FUNCTION_BLOCK sequence_T_08_loop (* Sequence with 8 Outputs looped, Transition by TIME *)
  (* Standard: 61499-2; Description: Copyright (c) 2024 HR Agrartechnik GmbH This program and the accompanying materials are made available under the terms of the Eclipse Public License 2.0 which is available at https://www.eclipse.org/legal/epl-2.0/ SPDX-License-Identifier: EPL-2.0 *)
  (* Version 1.0, 2024-03-02, Franz Höpfinger, HR Agrartechnik GmbH *)
  PACKAGE logiBUS::utils::sequence::timed;
  IMPORT logiBUS::utils::sequence::const::sequence;
  IMPORT logiBUS::utils::sequence::const::sequence::NO_TIME;
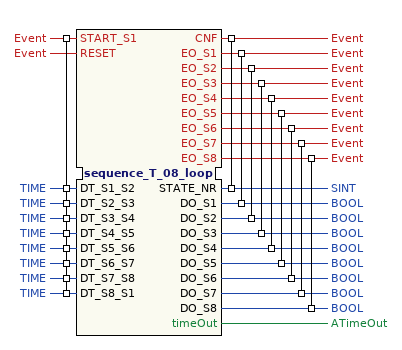
  EVENT_INPUT
    START_S1 WITH DT_S1_S2, DT_S2_S3, DT_S3_S4, DT_S4_S5, DT_S5_S6, DT_S6_S7, DT_S7_S8, DT_S8_S1; (* jump from START to State_01 *)
    RESET; (* Reset from any State to START *)
  END_EVENT
  EVENT_OUTPUT
    CNF WITH STATE_NR; (* Execution Confirmation *)
    EO_S1 WITH DO_S1;
    EO_S2 WITH DO_S2;
    EO_S3 WITH DO_S3;
    EO_S4 WITH DO_S4;
    EO_S5 WITH DO_S5;
    EO_S6 WITH DO_S6;
    EO_S7 WITH DO_S7;
    EO_S8 WITH DO_S8;
  END_EVENT
  VAR_INPUT
    DT_S1_S2 : TIME := NO_TIME; (* State_01 to State_02 timed *)
    DT_S2_S3 : TIME := NO_TIME; (* State_02 to State_03 timed *)
    DT_S3_S4 : TIME := NO_TIME; (* State_03 to State_04 timed *)
    DT_S4_S5 : TIME := NO_TIME; (* State_04 to State_05 timed *)
    DT_S5_S6 : TIME := NO_TIME; (* State_05 to State_06 timed *)
    DT_S6_S7 : TIME := NO_TIME; (* State_06 to State_07 timed *)
    DT_S7_S8 : TIME := NO_TIME; (* State_07 to State_08 timed *)
    DT_S8_S1 : TIME := NO_TIME; (* State_08 to State_01 timed *)
  END_VAR
  VAR_OUTPUT
    STATE_NR : SINT; (* State Number, START = 0, State_01 = 1 and so on. *)
    DO_S1 : BOOL; (* Output if State_01 is active *)
    DO_S2 : BOOL; (* Output if State_02 is active *)
    DO_S3 : BOOL; (* Output if State_03 is active *)
    DO_S4 : BOOL; (* Output if State_04 is active *)
    DO_S5 : BOOL; (* Output if State_05 is active *)
    DO_S6 : BOOL; (* Output if State_05 is active *)
    DO_S7 : BOOL; (* Output if State_05 is active *)
    DO_S8 : BOOL; (* Output if State_05 is active *)
  END_VAR
  PLUGS
    timeOut : iec61499::events::ATimeOut; (* timeOut Adapter *)
  END_PLUGS
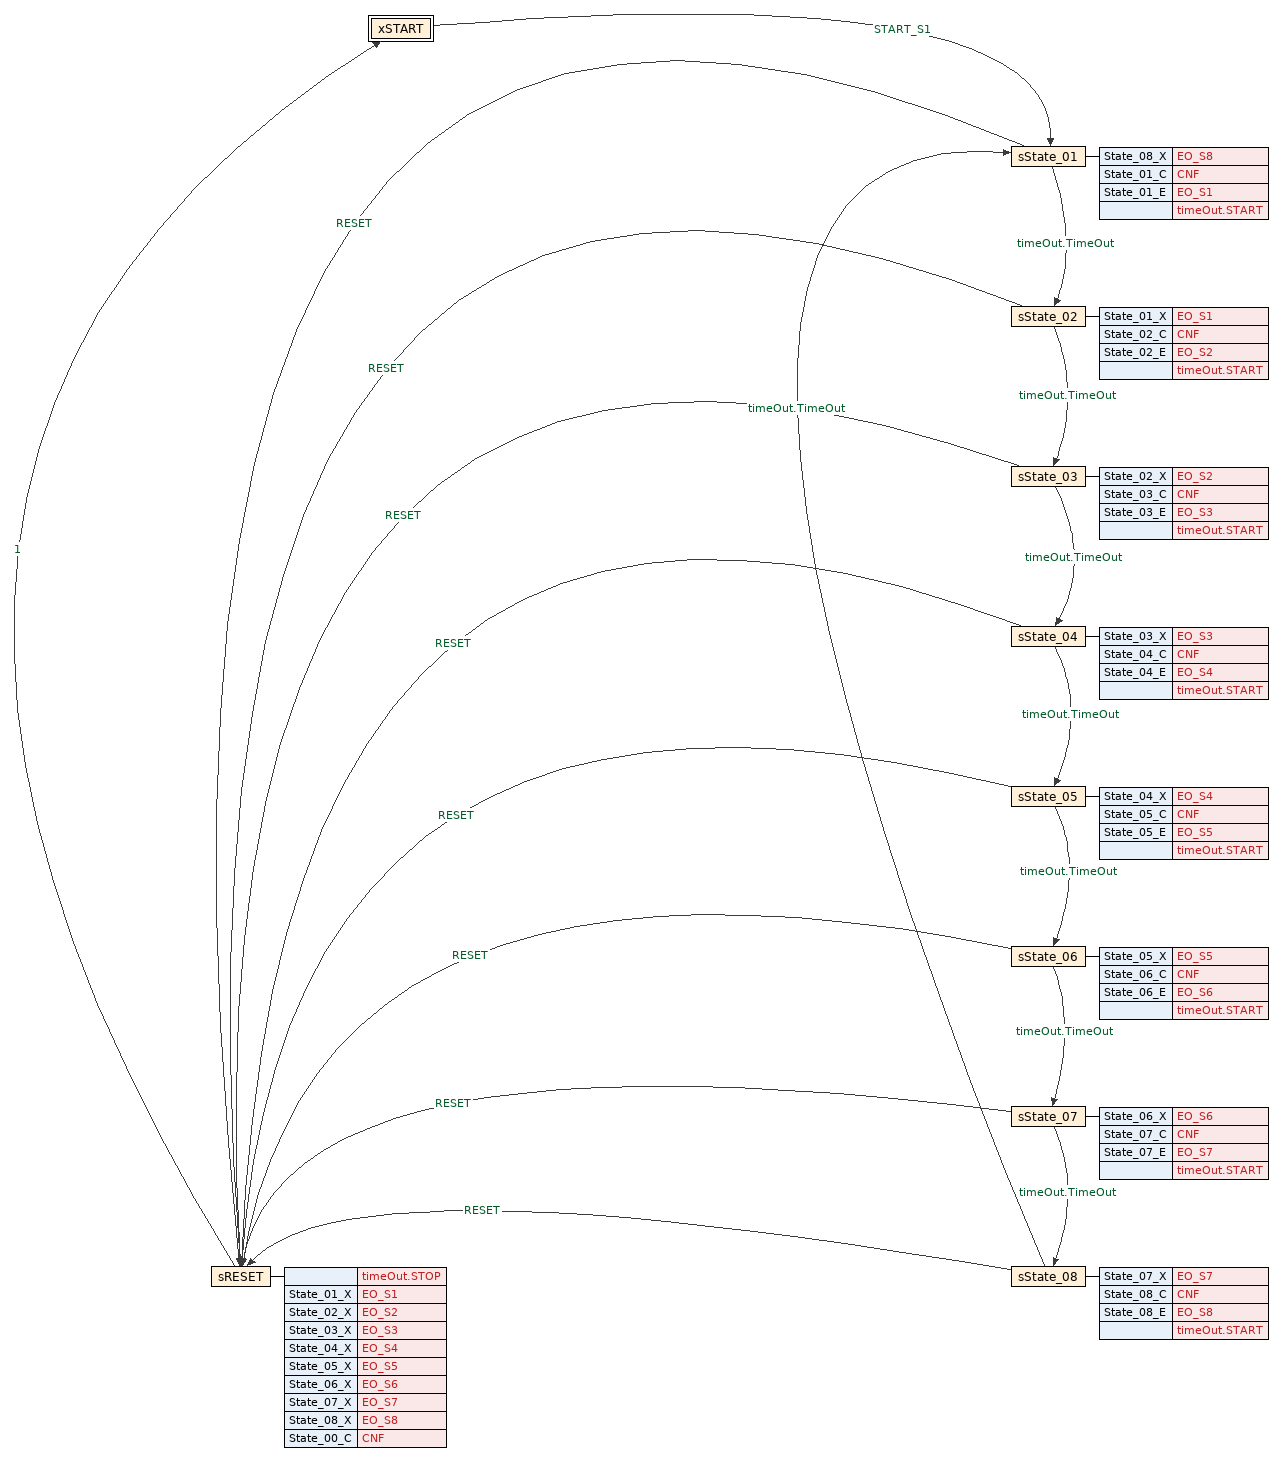
  EC_STATES
    xSTART; (* Initial State *)
    sState_01 : State_08_X -> EO_S8, State_01_C -> CNF, State_01_E -> EO_S1, -> timeOut.START;
    sState_02 : State_01_X -> EO_S1, State_02_C -> CNF, State_02_E -> EO_S2, -> timeOut.START;
    sState_03 : State_02_X -> EO_S2, State_03_C -> CNF, State_03_E -> EO_S3, -> timeOut.START;
    sState_04 : State_03_X -> EO_S3, State_04_C -> CNF, State_04_E -> EO_S4, -> timeOut.START;
    sState_05 : State_04_X -> EO_S4, State_05_C -> CNF, State_05_E -> EO_S5, -> timeOut.START;
    sState_06 : State_05_X -> EO_S5, State_06_C -> CNF, State_06_E -> EO_S6, -> timeOut.START;
    sState_07 : State_06_X -> EO_S6, State_07_C -> CNF, State_07_E -> EO_S7, -> timeOut.START;
    sState_08 : State_07_X -> EO_S7, State_08_C -> CNF, State_08_E -> EO_S8, -> timeOut.START;
    sRESET : -> timeOut.STOP, State_01_X -> EO_S1, State_02_X -> EO_S2, State_03_X -> EO_S3, State_04_X -> EO_S4, State_05_X -> EO_S5, State_06_X -> EO_S6, State_07_X -> EO_S7, State_08_X -> EO_S8, State_00_C -> CNF;
  END_STATES
  EC_TRANSITIONS
    sState_01 TO sState_02 := timeOut.TimeOut;
    sState_02 TO sState_03 := timeOut.TimeOut;
    sState_03 TO sState_04 := timeOut.TimeOut;
    xSTART TO sState_01 := START_S1;
    sState_01 TO sRESET := RESET;
    sState_02 TO sRESET := RESET;
    sState_03 TO sRESET := RESET;
    sState_04 TO sState_05 := timeOut.TimeOut;
    sState_04 TO sRESET := RESET;
    sState_05 TO sState_06 := timeOut.TimeOut;
    sState_05 TO sRESET := RESET;
    sState_07 TO sState_08 := timeOut.TimeOut;
    sState_07 TO sRESET := RESET;
    sState_06 TO sState_07 := timeOut.TimeOut;
    sState_06 TO sRESET := RESET;
    sRESET TO xSTART := 1;
    sState_08 TO sState_01 := timeOut.TimeOut;
    sState_08 TO sRESET := RESET;
  END_TRANSITIONS
  ALGORITHM State_00_C IN ST:
// Confirmation STEPS
// State_00 Confirmation Step
STATE_NR := sequence::State_00;
  END_ALGORITHM
  ALGORITHM State_01_C IN ST:
// State_01 Confirmation Step
STATE_NR := sequence::State_01;
timeOut.DT := DT_S1_S2;
  END_ALGORITHM
  ALGORITHM State_02_C IN ST:
// State_02 Confirmation Step
STATE_NR := sequence::State_02;
timeOut.DT := DT_S2_S3;
  END_ALGORITHM
  ALGORITHM State_03_C IN ST:
// State_03 Confirmation Step
STATE_NR := sequence::State_03;
timeOut.DT := DT_S3_S4;
  END_ALGORITHM
  ALGORITHM State_04_C IN ST:
// State_04 Confirmation Step
STATE_NR := sequence::State_04;
timeOut.DT := DT_S4_S5;
  END_ALGORITHM
  ALGORITHM State_05_C IN ST:
// State_05 Confirmation Step
STATE_NR := sequence::State_05;
timeOut.DT := DT_S5_S6;
  END_ALGORITHM
  ALGORITHM State_06_C IN ST:
// State_06 Confirmation Step
STATE_NR := sequence::State_06;
timeOut.DT := DT_S6_S7;
  END_ALGORITHM
  ALGORITHM State_07_C IN ST:
// State_07 Confirmation Step
STATE_NR := sequence::State_07;
timeOut.DT := DT_S7_S8;
  END_ALGORITHM
  ALGORITHM State_08_C IN ST:
// State_08 Confirmation Step
STATE_NR := sequence::State_08;
timeOut.DT := DT_S8_S1;
  END_ALGORITHM
  ALGORITHM State_01_E IN ST:
// State_01 Entry Step
DO_S1 := BOOL#TRUE; // ON
  END_ALGORITHM
  ALGORITHM State_01_X IN ST:
// State_01 Exit Step
DO_S1 := BOOL#FALSE;
  END_ALGORITHM
  ALGORITHM State_02_E IN ST:
// State_02 Entry Step
DO_S2 := BOOL#TRUE; // ON
  END_ALGORITHM
  ALGORITHM State_02_X IN ST:
// State_02 Exit Step
DO_S2 := BOOL#FALSE;
  END_ALGORITHM
  ALGORITHM State_03_E IN ST:
// State_03 Entry Step
DO_S3 := BOOL#TRUE; // ON
  END_ALGORITHM
  ALGORITHM State_03_X IN ST:
// State_03 Exit Step
DO_S3 := BOOL#FALSE;
  END_ALGORITHM
  ALGORITHM State_04_E IN ST:
// State_04 Entry Step
DO_S4 := BOOL#TRUE; // ON
  END_ALGORITHM
  ALGORITHM State_04_X IN ST:
// State_04 Exit Step
DO_S4 := BOOL#FALSE;
  END_ALGORITHM
  ALGORITHM State_05_E IN ST:
// State_05 Entry Step
DO_S5 := BOOL#TRUE; // ON
  END_ALGORITHM
  ALGORITHM State_05_X IN ST:
// State_05 Exit Step
DO_S5 := BOOL#FALSE;
  END_ALGORITHM
  ALGORITHM State_06_E IN ST:
// State_06 Entry Step
DO_S6 := BOOL#TRUE; // ON
  END_ALGORITHM
  ALGORITHM State_06_X IN ST:
// State_06 Exit Step
DO_S6 := BOOL#FALSE;
  END_ALGORITHM
  ALGORITHM State_07_E IN ST:
// State_07 Entry Step
DO_S7 := BOOL#TRUE; // ON
  END_ALGORITHM
  ALGORITHM State_07_X IN ST:
// State_07 Exit Step
DO_S7 := BOOL#FALSE;
  END_ALGORITHM
  ALGORITHM State_08_E IN ST:
// State_08 Entry Step
DO_S8 := BOOL#TRUE; // ON
  END_ALGORITHM
  ALGORITHM State_08_X IN ST:
// State_08 Exit Step
DO_S8 := BOOL#FALSE;
  END_ALGORITHM
END_FUNCTION_BLOCK
